(* CODESYS project Dry_Martini_System.project

Project tree, tasks and I/O mapping:
  Device : CODESYS Control Win V3, 3S - Smart Software Solutions GmbH, order no. 305021, version 3.5.6.10
    application Application
      libraries: Standard, * (System)
      task MainTask (cyclic, interval t#20ms, priority 1) calls Tester
      function block Totalizer [FBD]
      program Tester [LD]
      function block VCU [LD]
*)

// Device/Application/Tester
PROGRAM Tester
VAR
Vavula: BOOL;
LigaValvula: BOOL;
Abertura: TIME :=T#3S;



	LigaVvalvula: BOOL;
END_VAR

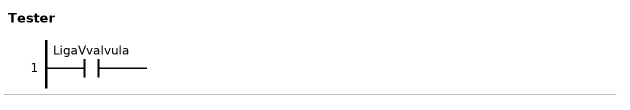
// NETWORK 1
(* LigaVvalvula; not connected *)

END_PROGRAM

// Device/Application/Totalizer
FUNCTION_BLOCK Totalizer
VAR_INPUT
	FlowRate: REAL; //vazão em L/s
	ValvIn: BOOL; //valvula anterior ao totalizador
	SavedCount: REAL; //valor armazenado
	TimeOpen: TIME; //tempo que a vávula permaneceu aberta
END_VAR
VAR_OUTPUT
	NewCount: REAL; //novo valor armazenado
END_VAR
VAR
	// Valor de contagem Parcial
	ParcialCount: REAL;
END_VAR

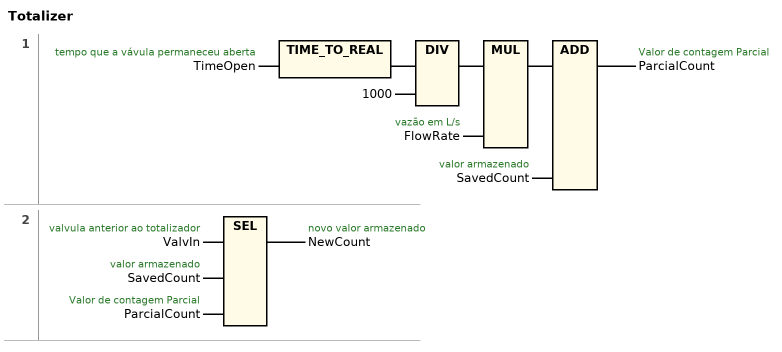
// NETWORK 1
//   TimeOpen: tempo que a vávula permaneceu aberta
//   FlowRate: vazão em L/s
//   SavedCount: valor armazenado
//   ParcialCount: Valor de contagem Parcial
ParcialCount := (TIME_TO_REAL(TimeOpen) / 1000) * FlowRate + SavedCount;

// NETWORK 2
//   ValvIn: valvula anterior ao totalizador
//   SavedCount: valor armazenado
//   ParcialCount: Valor de contagem Parcial
//   NewCount: novo valor armazenado
NewCount := SEL(ValvIn, SavedCount, ParcialCount);

END_FUNCTION_BLOCK

// Device/Application/VCU
FUNCTION_BLOCK VCU //Valv Controler Unit
VAR_INPUT
	TurnOn: BOOL; //comand to tunr on the valv
	FlowRate: REAL; //value of the floerate associated with the valv
	TimeOpen: TIME; //time indication, in seconds, that the valv need to be open 
END_VAR
VAR_OUTPUT
	Volume: REAL; //volume totalized 
	ValvState: BOOL; //indication of valv state (On or Off)
	
END_VAR
VAR
	TurnOff: BOOL; //turn off the valv
	SetVolume: BOOL; //alow the volumn total to be update
	TON_0: TON; //used to sutain the valv opening for the specified time
	Total1: Totalizer; //update the volume ctotal
	
END_VAR
VAR // added by the converter: edge detectors and wires of the graphical bodies
    _rt1 : R_TRIG;
END_VAR

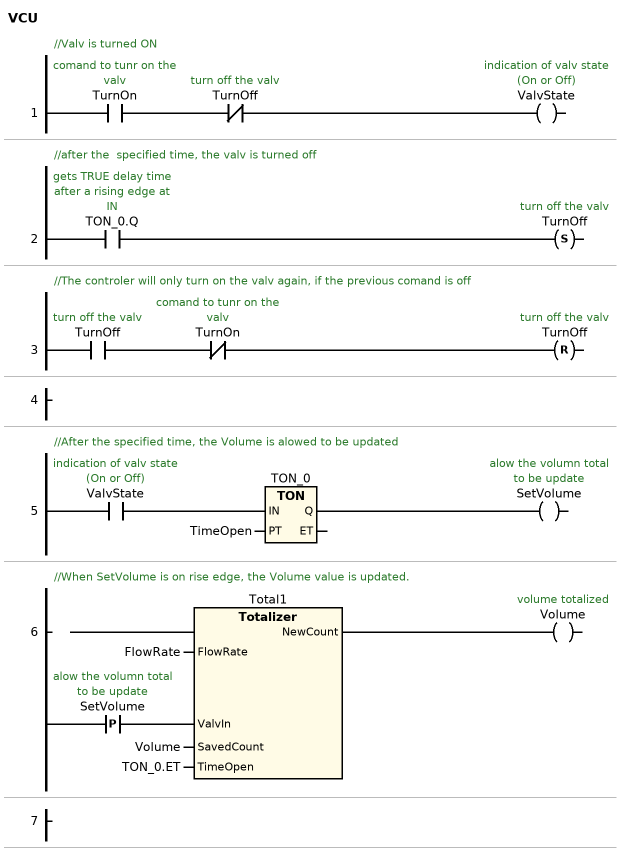
// NETWORK 1
// //Valv is turned ON
//   TurnOn: comand to tunr on the valv
//   TurnOff: turn off the valv
//   ValvState: indication of valv state (On or Off)
ValvState := TurnOn AND NOT TurnOff;

// NETWORK 2
// //after the  specified time, the valv is turned off
//   TON_0.Q: gets TRUE delay time after a rising edge at IN
//   TurnOff: turn off the valv
TurnOff S= TON_0.Q;

// NETWORK 3
// //The controler will only turn on the valv again, if the previous comand is off
//   TurnOff: turn off the valv
//   TurnOn: comand to tunr on the valv
TurnOff R= TurnOff AND NOT TurnOn;

// NETWORK 4

// NETWORK 5
// //After the specified time, the Volume is alowed to be updated
//   TON_0: used to sutain the valv opening for the specified time
//   ValvState: indication of valv state (On or Off)
//   TimeOpen: time indication, in seconds, that the valv need to be open
//   SetVolume: alow the volumn total to be update
TON_0(IN := ValvState, PT := TimeOpen); // TON
SetVolume := TON_0.Q;

// NETWORK 6
// //When SetVolume is on rise edge, the Volume value is updated.
//   Total1: update the volume ctotal
//   FlowRate: value of the floerate associated with the valv
//   SetVolume: alow the volumn total to be update
//   Volume: volume totalized
//   TON_0.ET: elapsed time since rising edge at IN
_rt1(CLK := SetVolume);
Total1(FlowRate := FlowRate, ValvIn := _rt1.Q, SavedCount := Volume, TimeOpen := TON_0.ET); // Totalizer
Volume := Total1.NewCount;

// NETWORK 7

END_FUNCTION_BLOCK
